(* PLC project Standard Funtion Blocks, Beremiz Additional Function Blocks Library 1.0, author Laurent Bessard *)
(* stored: creationDateTime 2013-09-09T09:56:11, modificationDateTime 2019-07-19T18:49:21 *)

(* The real time clock has many uses including time stamping, setting dates and times of day in batch reports, in alarm messages and so on. *)
FUNCTION_BLOCK RTC
  VAR_INPUT
    IN : BOOL;  (* 0 - current time, 1 - load time from PDT *)
    PDT : DT;  (* Preset datetime *)
  END_VAR
  VAR_OUTPUT
    Q : BOOL := FALSE;  (* Copy of IN *)
    CDT : DT;  (* Datetime, current or relative to PDT *)
  END_VAR
  VAR
    PREV_IN : BOOL := FALSE;
    OFFSET : TIME;
    CURRENT_TIME : DT;
  END_VAR

            {__SET_VAR(data__->,CURRENT_TIME,,__CURRENT_TIME)}

 IF IN
 THEN
   IF NOT PREV_IN
   THEN
       OFFSET := PDT - CURRENT_TIME;
   END_IF;

   (* PDT + time since PDT was loaded *)
   CDT := CURRENT_TIME + OFFSET;
 ELSE
   CDT := CURRENT_TIME;
 END_IF;

 Q := IN;
 PREV_IN := IN;

          
END_FUNCTION_BLOCK

(* The integral function block integrates the value of input XIN over time. *)
FUNCTION_BLOCK INTEGRAL
  VAR_INPUT
    RUN : BOOL;  (* 1 = integrate, 0 = hold *)
    R1 : BOOL;  (* Overriding reset *)
    XIN : REAL;  (* Input variable *)
    X0 : REAL;  (* Initial value *)
    CYCLE : TIME;  (* Sampling period *)
  END_VAR
  VAR_OUTPUT
    Q : BOOL;  (* NOT R1 *)
    XOUT : REAL;  (* Integrated output *)
  END_VAR

            Q := NOT R1 ;
IF R1 THEN XOUT := X0;
ELSIF RUN THEN XOUT := XOUT + XIN * TIME_TO_REAL(CYCLE);
END_IF;
          
END_FUNCTION_BLOCK

(* The derivative function block produces an output XOUT proportional to the rate of change of the input XIN. *)
FUNCTION_BLOCK DERIVATIVE
  VAR_INPUT
    RUN : BOOL;  (* 0 = reset *)
    XIN : REAL;  (* Input to be differentiated *)
    CYCLE : TIME;  (* Sampling period *)
  END_VAR
  VAR_OUTPUT
    XOUT : REAL;  (* Differentiated output *)
  END_VAR
  VAR
    X1 : REAL;
    X2 : REAL;
    X3 : REAL;
  END_VAR

            IF RUN THEN
  XOUT := (3.0 * (XIN - X3) + X1 - X2)
          / (10.0 * TIME_TO_REAL(CYCLE));
  X3 := X2;
  X2 := X1;
  X1 := XIN;
ELSE 
  XOUT := 0.0;
  X1 := XIN;
  X2 := XIN;
  X3 := XIN;
END_IF;
          
END_FUNCTION_BLOCK

(* The PID (proportional, Integral, Derivative) function block provides the classical three term controller for closed loop control. *)
FUNCTION_BLOCK PID
  VAR_INPUT
    AUTO : BOOL;  (* 0 - manual , 1 - automatic *)
    PV : REAL;  (* Process variable *)
    SP : REAL;  (* Set point *)
    X0 : REAL;  (* Manual output adjustment - Typically from transfer station *)
    KP : REAL;  (* Proportionality constant *)
    TR : REAL;  (* Reset time *)
    TD : REAL;  (* Derivative time constant *)
    CYCLE : TIME;  (* Sampling period *)
  END_VAR
  VAR_OUTPUT
    XOUT : REAL;
  END_VAR
  VAR
    ERROR : REAL;  (* PV - SP *)
    ITERM : INTEGRAL;  (* FB for integral term *)
    DTERM : DERIVATIVE;  (* FB for derivative term *)
  END_VAR

            ERROR := PV - SP ;
(*** Adjust ITERM so that XOUT := X0 when AUTO = 0 ***)
ITERM(RUN := AUTO, R1 := NOT AUTO, XIN := ERROR,
      X0 := TR * (X0 - ERROR), CYCLE := CYCLE);
DTERM(RUN := AUTO, XIN := ERROR, CYCLE := CYCLE);
XOUT := KP * (ERROR + ITERM.XOUT/TR + DTERM.XOUT*TD);
          
END_FUNCTION_BLOCK

(* The RAMP function block is modelled on example given in the standard. *)
FUNCTION_BLOCK RAMP
  VAR_INPUT
    RUN : BOOL;  (* 0 - track X0, 1 - ramp to/track X1 *)
    X0 : REAL;
    X1 : REAL;
    TR : TIME;  (* Ramp duration *)
    CYCLE : TIME;  (* Sampling period *)
  END_VAR
  VAR_OUTPUT
    BUSY : BOOL;  (* BUSY = 1 during ramping period *)
    XOUT : REAL := 0.0;
  END_VAR
  VAR
    XI : REAL;  (* Initial value *)
    T : TIME := T#0s;  (* Elapsed time of ramp *)
  END_VAR

            BUSY := RUN ;
IF RUN THEN
  IF T >= TR THEN 
    BUSY := 0;
    XOUT := X1;
  ELSE XOUT := XI + (X1-XI) * TIME_TO_REAL(T)
                            / TIME_TO_REAL(TR);
    T := T + CYCLE;
  END_IF;
ELSE
  XOUT := X0;
  XI := X0;
  T := T#0s;
END_IF;
          
END_FUNCTION_BLOCK

(* The hysteresis function block provides a hysteresis boolean output driven by the difference of two floating point (REAL) inputs XIN1 and XIN2. *)
FUNCTION_BLOCK HYSTERESIS
  VAR_INPUT
    XIN1 : REAL;
    XIN2 : REAL;
    EPS : REAL;
  END_VAR
  VAR_OUTPUT
    Q : BOOL;
  END_VAR

            IF Q THEN
  IF XIN1 < (XIN2 - EPS) THEN 
    Q := 0;
  END_IF;
ELSIF XIN1 > (XIN2 + EPS) THEN
  Q := 1;
END_IF;
          
END_FUNCTION_BLOCK
